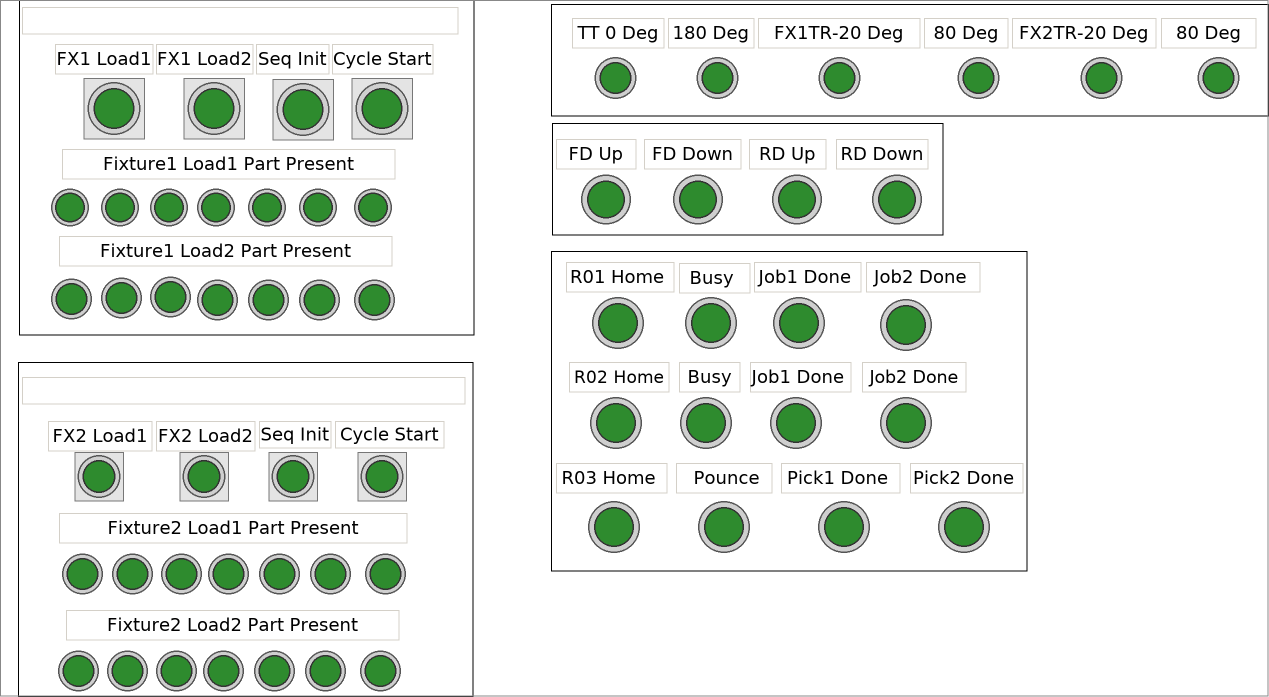
VISUALIZATION Fixture_Auto  // 1269x697
    Rectangle (18,362 455x335)
    Rectangle (19,0 455x335)
    Rectangle (551,4 718x112)
    Rectangle (552,123 391x112)
    Rectangle (551,251 476x320)
    Textfield (55,44 98x30), "FX1 Load1"
    Textfield (156,44 97x30), "FX1 Load2"
    PushSwitch (73,78 82x61), variable: Memory_DB.M_FX1_Load1, behaviour: TAP, style: Switch-PushSwitch-Green
    PushSwitch (173,78 82x61), variable: Memory_DB.M_FX1_Load2, behaviour: TAP, style: Switch-PushSwitch-Green
    Lamp1 (586,54 59x48), variable: Memory_DB.M_Turntable_POS1_Reached, style: Lamp-Lamp1-Green
    Textfield (572,18 92x30), "TT 0 Deg"
    Lamp1 (688,54 59x48), variable: Memory_DB.M_Turntable_POS2_Reached, style: Lamp-Lamp1-Green
    Textfield (668,18 86x30), "180 Deg"
    Textfield (256,44 73x30), "Seq Init"
    PushSwitch (262,79 82x61), variable: Memory_DB.M_FX1_All_Initialise, behaviour: TAP, style: Switch-PushSwitch-Green
    Lamp1 (810,54 59x48), variable: Memory_DB.M_Fixture1_TR_POS1_Reached, style: Lamp-Lamp1-Green
    Textfield (758,18 162x30), "FX1TR-20 Deg"
    Lamp1 (949,54 59x48), variable: Memory_DB.M_Fixture1_TR_POS2_Reached, style: Lamp-Lamp1-Green
    Textfield (924,18 84x30), "80 Deg"
    Lamp1 (571,171 70x57), variable: Inputs.i_Front_Door_Up, style: Lamp-Lamp1-Green
    Textfield (556,139 80x30), "FD Up"
    Lamp1 (663,171 70x57), variable: Inputs.i_Front_Door_Down, style: Lamp-Lamp1-Green
    Textfield (644,139 97x30), "FD Down"
    Lamp1 (762,171 70x57), variable: Inputs.i_Rear_Door_Up, style: Lamp-Lamp1-Green
    Textfield (749,139 77x30), "RD Up"
    Lamp1 (862,171 70x57), variable: Inputs.i_Rear_Door_Down, style: Lamp-Lamp1-Green
    Textfield (836,139 92x30), "RD Down"
    Lamp1 (588,293 60x60), variable: Memory_DB.M_R01_Home, style: Lamp-Lamp1-Green
    Textfield (566,262 108x30), "R01 Home"
    Lamp1 (769,293 60x60), variable: Memory_DB.M_R01_Job_Done1, style: Lamp-Lamp1-Green
    Textfield (754,262 107x30), "Job1 Done"
    Lamp1 (586,393 60x60), variable: Memory_DB.M_R02_Home, style: Lamp-Lamp1-Green
    Textfield (569,362 100x30), "R02 Home"
    Lamp1 (766,393 60x60), variable: Memory_DB.M_R02_Job_Done1, style: Lamp-Lamp1-Green
    Textfield (750,362 101x30), "Job1 Done"
    Lamp1 (579,497 70x60), variable: Memory_DB.M_R03_MH_AtHome, style: Lamp-Lamp1-Green
    Textfield (556,463 111x30), "R03 Home"
    Lamp1 (689,497 70x60), variable: Memory_DB.M_R03_MH_AtPounce, style: Lamp-Lamp1-Green
    Textfield (676,463 96x30), "Pounce"
    Lamp1 (929,497 70x60), variable: Memory_DB.M_R03_MH_Pick2_Done, style: Lamp-Lamp1-Green
    Textfield (910,463 113x30), "Pick2 Done"
    Lamp1 (809,497 70x60), variable: Memory_DB.M_R03_MH_Pick1_Done, style: Lamp-Lamp1-Green
    Textfield (781,463 119x30), "Pick1 Done"
    Lamp1 (48,184 44x47), variable: Inputs.i_FX1_PART_CONTROL_B1, style: Lamp-Lamp1-Green
    Textfield (62,149 333x30), "Fixture1 Load1 Part Present"
    Lamp1 (98,184 44x47), variable: Inputs.i_FX1_PART_CONTROL_B2, style: Lamp-Lamp1-Green
    Lamp1 (147,184 44x47), variable: Inputs.i_FX1_PART_CONTROL_B3, style: Lamp-Lamp1-Green
    Lamp1 (194,184 44x47), variable: Inputs.i_FX1_PART_CONTROL_B4, style: Lamp-Lamp1-Green
    Lamp1 (245,184 44x47), variable: Inputs.i_FX1_PART_CONTROL_B5, style: Lamp-Lamp1-Green
    Lamp1 (296,184 44x47), variable: Inputs.i_FX1_PART_CONTROL_B6, style: Lamp-Lamp1-Green
    Lamp1 (351,184 44x47), variable: Inputs.i_FX1_PART_CONTROL_B7, style: Lamp-Lamp1-Green
    Lamp1 (48,273 47x52), variable: Inputs.i_FX1_PART_CONTROL_B15, style: Lamp-Lamp1-Green
    Textfield (59,236 333x30), "Fixture1 Load2 Part Present"
    Lamp1 (98,272 47x52), variable: Inputs.i_FX1_PART_CONTROL_B16, style: Lamp-Lamp1-Green
    Lamp1 (147,271 47x52), variable: Inputs.i_FX1_PART_CONTROL_B17, style: Lamp-Lamp1-Green
    Lamp1 (194,274 47x52), variable: Inputs.i_FX1_PART_CONTROL_B18, style: Lamp-Lamp1-Green
    Lamp1 (245,274 47x52), variable: Inputs.i_FX1_PART_CONTROL_B19, style: Lamp-Lamp1-Green
    Lamp1 (296,274 47x52), variable: Inputs.i_FX1_PART_CONTROL_B20, style: Lamp-Lamp1-Green
    Lamp1 (351,274 47x52), variable: Inputs.i_FX1_PART_CONTROL_B21, style: Lamp-Lamp1-Green
    Lamp1 (876,295 60x60), variable: Memory_DB.M_R01_Job_Done2, style: Lamp-Lamp1-Green
    Textfield (866,262 114x30), "Job2 Done"
    Lamp1 (876,393 60x60), variable: Memory_DB.M_R02_Job_Done2, style: Lamp-Lamp1-Green
    Textfield (862,362 104x30), "Job2 Done"
    Lamp1 (676,393 60x60), variable: Memory_DB.M_R02_Busy, style: Lamp-Lamp1-Green
    Lamp1 (681,293 60x60), variable: Memory_DB.M_R01_Busy, style: Lamp-Lamp1-Green
    Textfield (679,263 71x30), "Busy"
    Textfield (679,362 61x30), "Busy"
    Textfield (332,44 101x30), "Cycle Start"
    PushSwitch (341,78 82x61), variable: Memory_DB.M_FX1_Cycle_Start_PB, behaviour: TAP, style: Switch-PushSwitch-Green
    Textfield (48,421 104x30), "FX2 Load1"
    Textfield (156,421 99x30), "FX2 Load2"
    PushSwitch (67,452 64x49), variable: Memory_DB.M_FX2_Load1, behaviour: TAP, style: Switch-PushSwitch-Green
    PushSwitch (172,452 64x49), variable: Memory_DB.M_FX2_Load2, behaviour: TAP, style: Switch-PushSwitch-Green
    Textfield (259,421 72x27), "Seq Init"
    PushSwitch (261,452 64x49), variable: Memory_DB.M_FX2_All_Initialise, behaviour: TAP, style: Switch-PushSwitch-Green
    Lamp1 (59,548 47x52), variable: Inputs.i_FX2_PART_CONTROL_B1, style: Lamp-Lamp1-Green
    Textfield (59,513 348x30), "Fixture2 Load1 Part Present"
    Lamp1 (109,548 47x52), variable: Inputs.i_FX2_PART_CONTROL_B2, style: Lamp-Lamp1-Green
    Lamp1 (158,548 47x52), variable: Inputs.i_FX2_PART_CONTROL_B3, style: Lamp-Lamp1-Green
    Lamp1 (205,548 47x52), variable: Inputs.i_FX2_PART_CONTROL_B4, style: Lamp-Lamp1-Green
    Lamp1 (256,548 47x52), variable: Inputs.i_FX2_PART_CONTROL_B5, style: Lamp-Lamp1-Green
    Lamp1 (307,548 47x52), variable: Inputs.i_FX2_PART_CONTROL_B6, style: Lamp-Lamp1-Green
    Lamp1 (362,548 47x52), variable: Inputs.i_FX2_PART_CONTROL_B7, style: Lamp-Lamp1-Green
    Lamp1 (55,645 47x52), variable: Inputs.i_FX2_PART_CONTROL_B15, style: Lamp-Lamp1-Green
    Textfield (66,610 333x30), "Fixture2 Load2 Part Present"
    Lamp1 (104,645 47x52), variable: Inputs.i_FX2_PART_CONTROL_B16, style: Lamp-Lamp1-Green
    Lamp1 (153,645 47x52), variable: Inputs.i_FX2_PART_CONTROL_B17, style: Lamp-Lamp1-Green
    Lamp1 (200,645 47x52), variable: Inputs.i_FX2_PART_CONTROL_B18, style: Lamp-Lamp1-Green
    Lamp1 (251,645 47x52), variable: Inputs.i_FX2_PART_CONTROL_B19, style: Lamp-Lamp1-Green
    Lamp1 (302,645 47x52), variable: Inputs.i_FX2_PART_CONTROL_B20, style: Lamp-Lamp1-Green
    Lamp1 (357,645 47x52), variable: Inputs.i_FX2_PART_CONTROL_B21, style: Lamp-Lamp1-Green
    Lamp1 (1072,54 59x48), variable: Memory_DB.M_Fixture2_TR_POS1_Reached, style: Lamp-Lamp1-Green
    Textfield (1012,18 144x30), "FX2TR-20 Deg"
    Lamp1 (1189,54 59x48), variable: Memory_DB.M_Fixture2_TR_POS2_Reached, style: Lamp-Lamp1-Green
    Textfield (1161,18 95x30), "80 Deg"
    PushSwitch (350,452 64x49), variable: Memory_DB.M_FX2_Cycle_Start_PB, behaviour: TAP, style: Switch-PushSwitch-Green
    Textfield (335,421 109x27), "Cycle Start"
    Textfield (22,7 436x27), text list: 'FX1TextList', text index: Fixture1_Auto.nState_Door
    Textfield (22,377 443x27), text list: 'FX2TextList', text index: Fixture2_Auto.nState_Door
END_VISUALIZATION

(* stored: Version 1.1.0.1, ProductVersion 3.1.4024.16
   Visu Fixture_Auto: Id {79b35ba8-3b90-46a6-8c72-63d1c4694cd8} *)
